{attribute addProperty BoxType "ELM2642-0000-0016"}
{attribute addProperty Id "Outputs_Channel_1AT %Q*Outputs_Channel_E6FE5E20162"}
{attribute addProperty CRC "2975667360"}
{attribute addProperty SizeInBites "16"}
{attribute addProperty SizeInBytes "2"}
TYPE DO_Group_1_Outputs_B15D14A0 :
STRUCT
	{attribute addProperty Name "Outputs_Channel_1"}
	Outputs_Channel_1 AT %Q* : Outputs_Channel_E6FE5E20;
END_STRUCT
END_TYPE

(* stored: Version 1.2.0.0, ProductVersion 3.1.4024.9
   DUT DO_Group_1_Outputs_B15D14A0: Id {5a03ba82-b5b6-4cf2-aff4-f4389ab4ac69} *)
